// TIA Portal V20 export
ORGANIZATION_BLOCK "Startup"   // OB1050, LAD, Startup
TITLE = "Complete Restart"
// stored: AutoNumber false, Namespace Unit1.Em9, SetENOAutomatically false
   VAR_INPUT
      LostRetentive : Bool;   // True if retentive data are lost
      LostRTC : Bool;   // True if date and time are lost
   END_VAR
BEGIN

REGION Network 1 (SCL): Build the Absolut Reference Designator
   // Set the Absoult Reference Designator in the Config DB
   IF LEN(IN := "Unit1.Em9.Config".em.referenceDesignator.parent) <> 0 THEN
       "Unit1.Em9.Config".em.referenceDesignator.combined := CONCAT_WSTRING(IN1 := "Unit1.Em9.Config".em.referenceDesignator.parent, IN2 := WSTRING#'.', IN3 := "Unit1.Em9.Config".em.referenceDesignator.relative);
   ELSE
       "Unit1.Em9.Config".em.referenceDesignator.combined := "Unit1.Em9.Config".em.referenceDesignator.relative;
   END_IF;
END_REGION
END_ORGANIZATION_BLOCK
